TYPE CmpWorkStopMainLnSwSim :
STRUCT
	DBBypass: BOOL;
	ForceRFID: BOOL;
	TestRFIDData: DINT := 404;
	TestPuckData: DBGetOutputLane;
END_STRUCT
END_TYPE

(* stored: Version 1.1.0.1, ProductVersion 3.1.4024.6
   DUT CmpWorkStopMainLnSwSim: Id {0dc07ba5-3ad4-4aef-967d-52b265b718bc} *)
